# EPICS substitutions: evrIoc/Db/evrPatternXL04.substitutions
#
# Pattern records
file evrPatternAll.db
{
  pattern { DEVICE        , LINK4 ,  LINK5                    ,        LINK6                  , TREF , TS1ST, TS2ND }
	  { IOC:XL04:EV01 ,  ""   , "IOC:XL04:EV01:FANOUT PP" , "ESIM:XL04:1:PATTERNSIMFO PP" , 1E06 ,   1  ,   4   }
}
file evrPatternTest.db
{
pattern { DEVICE        , SIMUL       }
        { IOC:XL04:EV01 , ESIM:XL04:1 }
}
file evrPatternProc_event.db
{
pattern {    DEV          }
        { "IOC:XL04:EV01" }
}
